FUNCTION_BLOCK FB_LimSwStatus_testDouble IMPLEMENTS I_LimSwStatus
VAR
   // NC Forward Limit Switch: TRUE if ok to move
    bLimitForwardEnable : BOOL := TRUE;
    // NC Backward Limit Switch: TRUE if ok to move
    bLimitBackwardEnable : BOOL := TRUE;
    // NO Home Switch: TRUE if at home
    bHome : BOOL;
END_VAR

PROPERTY LimBackward : BOOL
GET
LimBackward := bLimitBackwardEnable;
END_GET
SET
bLimitBackwardEnable := LimBackward;
END_SET
END_PROPERTY

PROPERTY LimForward : BOOL
GET
LimForward := bLimitForwardEnable;
END_GET
SET
bLimitForwardEnable := LimForward;
END_SET
END_PROPERTY

PROPERTY LimHome : BOOL
GET
 LimHome := bHome;
END_GET
SET
 bHome := LimHome;
END_SET
END_PROPERTY

END_FUNCTION_BLOCK

(* stored: Version 1.1.0.1
   POU FB_LimSwStatus_testDouble: Id {70960280-1575-4989-a963-b01a3910fbdc}, SpecialFunc None
   Property LimBackward: Id {28e716fb-4cd1-40e4-8576-b647717a5062}
   Get Get: Id {b69eedf2-23f9-4507-93d5-1b56ab38615d}
   Set Set: Id {96af2482-9e4a-46c5-954f-4aa47f4efe5b}
   Property LimForward: Id {94d01c11-2835-4a77-869c-e37196b02038}
   Get Get: Id {dcbc549b-c86c-4198-ad11-9e83448e0922}
   Set Set: Id {55b3cb2d-deb6-4811-a76c-1c504a6f46c0}
   Property LimHome: Id {e76f8bd1-7a05-4eac-bf90-76b44ef399a2}
   Get Get: Id {a49f8d60-57a6-4b05-b188-1b8613fd3fb4}
   Set Set: Id {2cf8e61a-e230-43f8-95fa-8485ce107d19} *)
